TYPE csp_case_feed_reject_sensors_status_enum :
(
	IN_RANGE1 			:= 0,
	OUT_OF_LOWER_RANGE1 := 1,
	OUT_OF_UPPER_RANGE1 := 2,
	NOT_CHECKED1 		:= 10
) := NOT_CHECKED1;
END_TYPE

(* stored: Version 1.1.0.1, ProductVersion 3.1.4024.3
   DUT csp_case_feed_reject_sensors_status_enum: Id {2c26bdd3-b212-4c6a-bc16-ae4ee0072dde} *)
